FUNCTION TFPackCodePresenteInWAJolly : INT
VAR_INPUT
	//HandlingPackTable : POINTER TO TFHandlingPackTable;
	ArrayPacchi : POINTER TO DUT_ArrayPacchi;
	WorkArea : POINTER TO ARRAY [1..MAXAREA] OF TFMachinePalletizer_WorkArea;
	WorkAreaState : POINTER TO ARRAY [1..MAXAREA] OF TFMachinePalletizer_WorkAreaState;
END_VAR
VAR
	w : INT;
	wa : INT;
	i : INT;
END_VAR

TFPackCodePresenteInWAJolly := 0; 

FOR w:=MAXDIMARRAYPACCHI TO 1 BY -1 DO
	IF ArrayPacchi^.Pacco[w].PC > 0 THEN
		FOR wa:=1 TO MAXAREA DO
			IF WorkArea^[wa].Code = ArrayPacchi^.Pacco[w].PC THEN
				(* Verifico se la piazzola è in lavorazione *)
				(* Se è in lavorazione allora è inutile assegnarne un'altra con lo stesso codice *)
				IF WorkAreaState^[wa].State < WORKAREA_STATE_OCCUPIED_WORKED THEN
					TFPackCodePresenteInWAJolly := 0;
					RETURN;
				//ELSE
					//TFPackCodePresentToJollyWorkArea := WorkPickPointState^[w].Code;
				END_IF
				//RETURN;
			END_IF
		END_FOR
		TFPackCodePresenteInWAJolly := ArrayPacchi^.Pacco[w].PC;
	END_IF	
END_FOR

END_FUNCTION

(* stored: Version 1.1.0.1, ProductVersion 3.1.4024.11
   POU TFPackCodePresenteInWAJolly: Id {d604903e-034f-4697-be43-951227e30fc9}, SpecialFunc None *)
